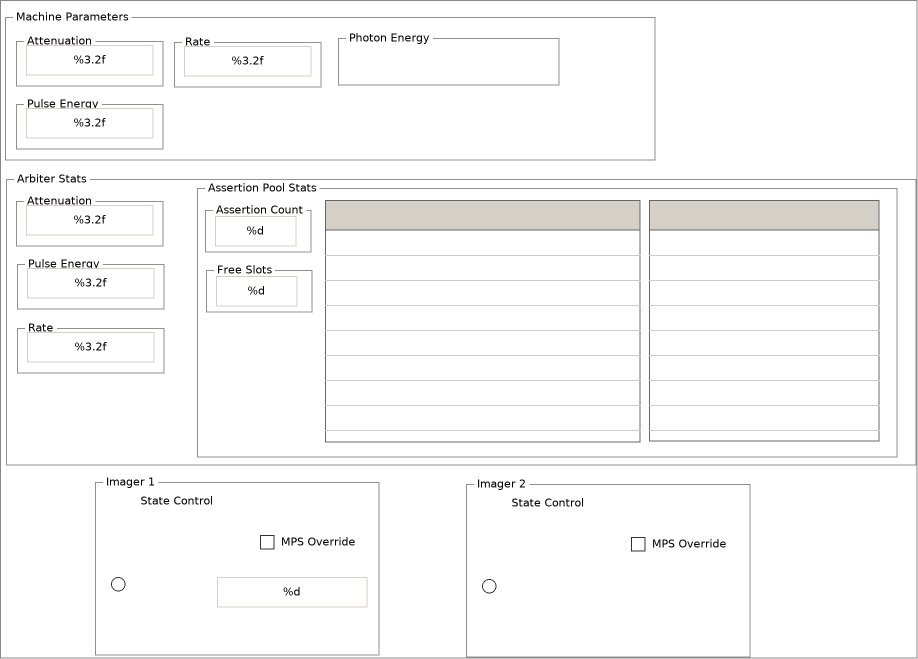
VISUALIZATION Visualization  // 918x659
    GroupBox (5,9 650x151), "Machine Parameters"
        GroupBox (11,24 147x53), "Attenuation"
            Textfield (10,12 127x30), "%3.2f", text variable: PMPS_GVL_BeamParams.stCurrentBeamParameters.fAtt
        GroupBox (11,87 147x53), "Pulse Energy"
            Textfield (10,12 127x30), "%3.2f", text variable: PMPS_GVL_BeamParams.stCurrentBeamParameters.fPP_mJ
        GroupBox (169,25 147x53), "Rate"
            Textfield (10,12 127x30), "%3.2f", text variable: PMPS_GVL_BeamParams.stCurrentBeamParameters.nRate
        GroupBox (333,21 221x55), "Photon Energy"
    GroupBox (6,171 910x294), "Arbiter Stats"
        GroupBox (191,9 700x277), "Assertion Pool Stats"
            GroupBox (9,82 106x50), "Free Slots"
                Textfield (10,14 81x30), "%d", text variable: fbArbiter.fbBPAssertionPool.hTable.nFree
            GroupBox (8,22 106x50), "Assertion Count"
                Textfield (10,14 81x30), "%d", text variable: fbArbiter.fbBPAssertionPool.hTable.nCount
            Table (128,20 315x242), data array: fbArbiter.fbBPAssertionPool.dataPool
                p3854506369: fbArbiter.fbBPAssertionPool.dataPool[INDEX].fAtt
                p1892666644: fbArbiter.fbBPAssertionPool.dataPool[INDEX].fPP_mJ
                p338671338: fbArbiter.fbBPAssertionPool.dataPool[INDEX].fUpper_eV
                p2170511999: fbArbiter.fbBPAssertionPool.dataPool[INDEX].fLower_eV
                p1755163831: Upper eV
                p4092479075: Lower eV
            Table (452,20 230x241), data array: fbArbiter.fbBPAssertionPool.entries
                p3854506369: fbArbiter.fbBPAssertionPool.entries[INDEX].key
                p1892666644: fbArbiter.fbBPAssertionPool.entries[INDEX].value
                p338671338: fbArbiter.fbBPAssertionPool.entries[INDEX].lock
                p2170511999: fbArbiter.fbBPAssertionPool.entries[INDEX].pNext
                p3723444502: fbArbiter.fbBPAssertionPool.entries[INDEX].pNextFree
                p1218418051: fbArbiter.fbBPAssertionPool.entries[INDEX].pNextGlob
                p2232123230: Assertion ID
        GroupBox (10,22 147x53), "Attenuation"
            Textfield (10,12 127x30), "%3.2f", text variable: fbArbiter.q_stBeamParams.fAtt
        GroupBox (11,85 147x53), "Pulse Energy"
            Textfield (10,12 127x30), "%3.2f", text variable: fbArbiter.q_stBeamParams.fPP_mJ
        GroupBox (11,149 147x53), "Rate"
            Textfield (10,12 127x30), "%3.2f", text variable: fbArbiter.stOutputBP.nRate
    GroupBox (466,476 284x181), "Imager 2"
        RadioButton (14,49 97x122), variable: MAIN.fbDev2.stDevice.nRequestedState
            Areas[1]: Text=State 1
            Areas[2]: Text=State 2
            Areas[3]: Text=State 3
        Label (7,12 150x30), "State Control"
        Checkbox (163,53 110x30), "MPS Override", variable: MAIN.fbDev2.stDevice.xOverrideMPSLimits
    GroupBox (95,474 284x181), "Imager 1"
        RadioButton (14,49 97x122), variable: MAIN.fbDev1.stDevice.nRequestedState
            Areas[1]: Text=State 1
            Areas[2]: Text=State 2
            Areas[3]: Text=State 3
        Label (7,12 150x30), "State Control"
        Checkbox (163,53 111x30), "MPS Override", variable: MAIN.fbDev1.stDevice.xOverrideMPSLimits
        Textfield (122,103 150x30), "%d", text variable: MAIN.fbDev1.stDevice.nRequestedState
            OnMouseClick: write the text variable via Default
END_VISUALIZATION

(* stored: Version 1.1.0.1, ProductVersion 3.1.4022.12
   Visu Visualization: Id {e2d11be7-f40a-0a2a-160a-0d1b47b9df45} *)
